{attribute 'qualified_only'}
{attribute 'strict'}
TYPE E_Mode :
(
	Off := 1,
	Manual := 0,
	Auto := 0
);
END_TYPE

(* stored: Version 1.1.0.1, ProductVersion 3.1.4024.9
   DUT E_Mode: Id {16394d50-8d60-4125-b4f7-3915c90f53a5} *)
